// TIA Portal V20 export
TYPE "UDT_PowermeterMeasure"
   STRUCT
      NbMeasure : Int := 100;
      ActualMeasure : Int;
      ActualTotalMeas : Real;
      Table_full : Bool;   // TRUE when the table are fully of measures
      Measures : Array[0..99] of Struct
         Time_day : Time_Of_Day;
         Day_meas : Date;
         Job_meas : Int;
         ValuePower : Real;
         ValueCM : Real;
      END_STRUCT;
   END_STRUCT;
END_TYPE
